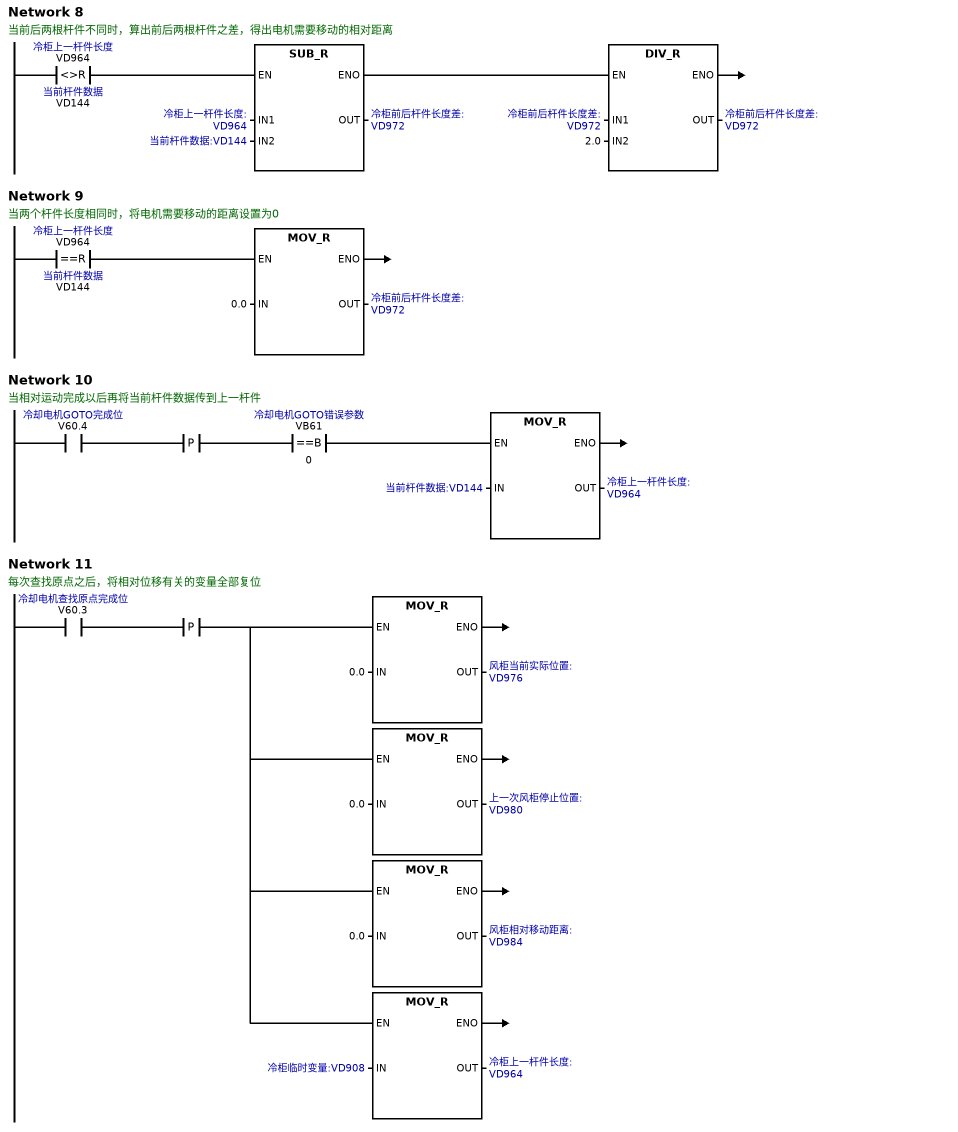
[picture p24: SBR16 networks 8-11]
Network 8
// 当前后两根杆件不同时，算出前后两根杆件之差，得出电机需要移动的相对距离
LDR<>  冷柜上一杆件长度:VD964, 当前杆件数据:VD144
MOVR   冷柜上一杆件长度:VD964, 冷柜前后杆件长度差:VD972
AENO
-R     当前杆件数据:VD144, 冷柜前后杆件长度差:VD972
AENO
/R     2.0, 冷柜前后杆件长度差:VD972
Network 9
// 当两个杆件长度相同时，将电机需要移动的距离设置为0
LDR=   冷柜上一杆件长度:VD964, 当前杆件数据:VD144
MOVR   0.0, 冷柜前后杆件长度差:VD972
Network 10
// 当相对运动完成以后再将当前杆件数据传到上一杆件
LD     冷却电机GOTO完成位:V60.4
EU
AB=    冷却电机GOTO错误参数:VB61, 0
MOVR   当前杆件数据:VD144, 冷柜上一杆件长度:VD964
Network 11
// 每次查找原点之后，将相对位移有关的变量全部复位
LD     冷却电机查找原点完成位:V60.3
EU
MOVR   0.0, 风柜当前实际位置:VD976
MOVR   0.0, 上一次风柜停止位置:VD980
MOVR   0.0, 风柜相对移动距离:VD984
MOVR   冷柜临时变量:VD908, 冷柜上一杆件长度:VD964
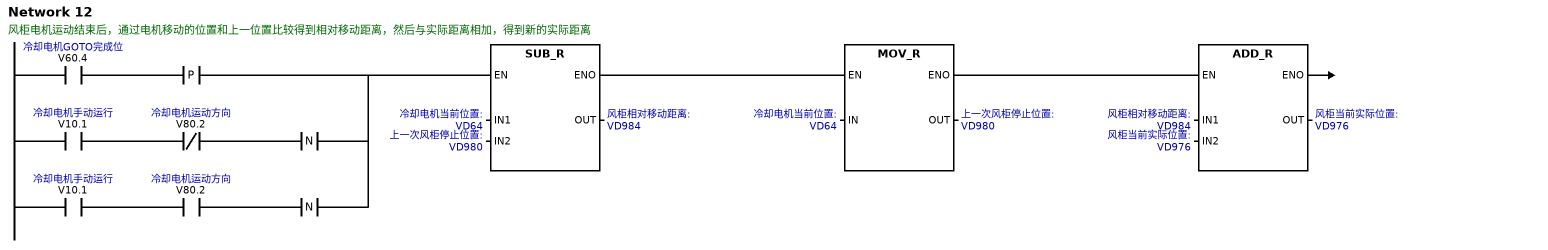
Network 12
// 风柜电机运动结束后，通过电机移动的位置和上一位置比较得到相对移动距离，然后与实际距离相加，得到新的实际距离
LD     冷却电机GOTO完成位:V60.4
EU
LD     冷却电机手动运行:V10.1
AN     冷却电机运动方向:V80.2
ED
OLD
LD     冷却电机手动运行:V10.1
A      冷却电机运动方向:V80.2
ED
OLD
MOVR   冷却电机当前位置:VD64, 风柜相对移动距离:VD984
AENO
-R     上一次风柜停止位置:VD980, 风柜相对移动距离:VD984
AENO
MOVR   冷却电机当前位置:VD64, 上一次风柜停止位置:VD980
AENO
+R     风柜相对移动距离:VD984, 风柜当前实际位置:VD976
END_SUBROUTINE_BLOCK

SUBROUTINE_BLOCK 冷却电机手动控制:SBR18
TITLE=子程序注释
BEGIN
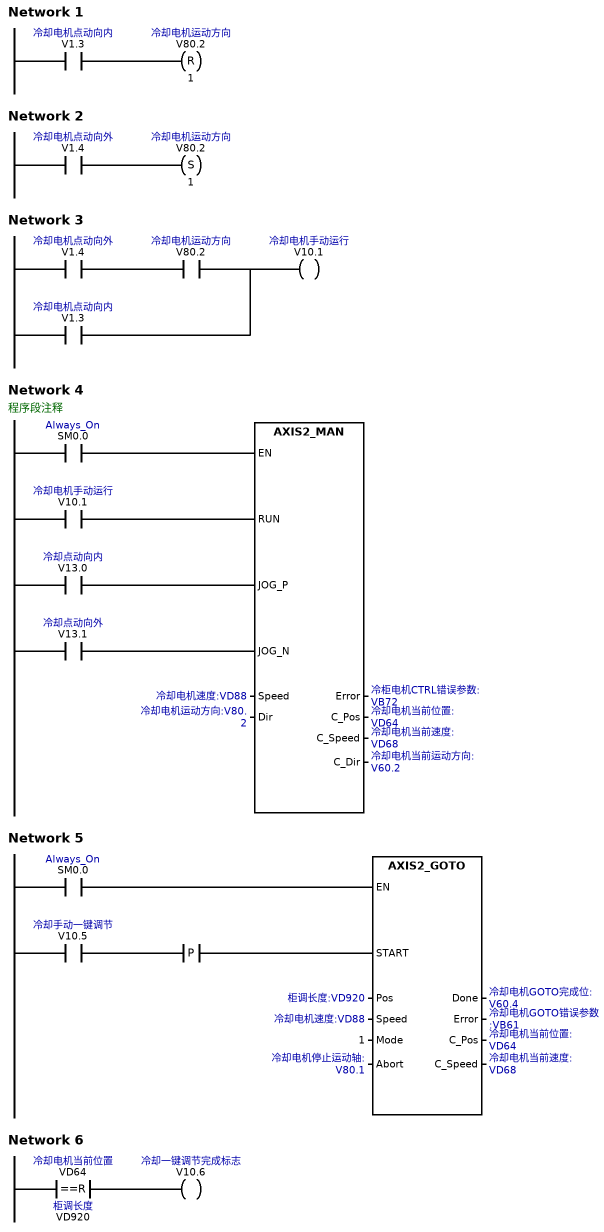
Network 1
LD     冷却电机点动向内:V1.3
R      冷却电机运动方向:V80.2, 1
Network 2
LD     冷却电机点动向外:V1.4
S      冷却电机运动方向:V80.2, 1
Network 3
LD     冷却电机点动向外:V1.4
A      冷却电机运动方向:V80.2
O      冷却电机点动向内:V1.3
=      冷却电机手动运行:V10.1
Network 4
// 程序段注释
LD     Always_On:SM0.0
=      L60.0
LD     冷却电机手动运行:V10.1
=      L63.7
LD     冷却点动向内:V13.0
=      L63.6
LD     冷却点动向外:V13.1
=      L63.5
LD     L60.0
CALL   AXIS2_MAN:SBR11, L63.7, L63.6, L63.5, 冷却电机速度:VD88, 冷却电机运动方向:V80.2, 冷柜电机CTRL错误参数:VB72, 冷却电机当前位置:VD64, 冷却电机当前速度:VD68, 冷却电机当前运动方向:V60.2
Network 5
LD     Always_On:SM0.0
=      L60.0
LD     冷却手动一键调节:V10.5
EU
=      L63.7
LD     L60.0
CALL   AXIS2_GOTO:SBR12, L63.7, 柜调长度:VD920, 冷却电机速度:VD88, 1, 冷却电机停止运动轴:V80.1, 冷却电机GOTO完成位:V60.4, 冷却电机GOTO错误参数:VB61, 冷却电机当前位置:VD64, 冷却电机当前速度:VD68
Network 6
LDR=   冷却电机当前位置:VD64, 柜调长度:VD920
=      冷却一键调节完成标志:V10.6
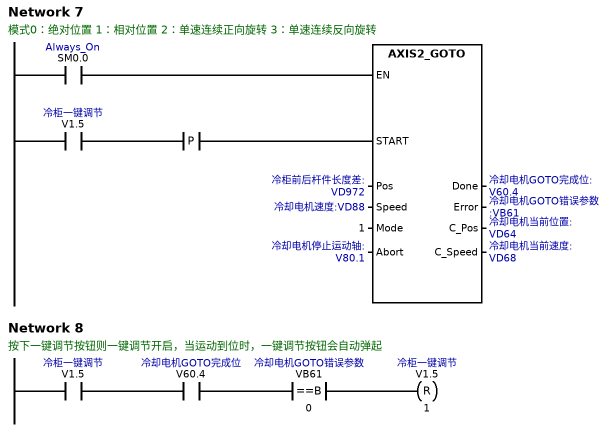
Network 7
// 模式0：绝对位置 1：相对位置 2：单速连续正向旋转 3：单速连续反向旋转
LD     Always_On:SM0.0
=      L60.0
LD     冷柜一键调节:V1.5
EU
=      L63.7
LD     L60.0
CALL   AXIS2_GOTO:SBR12, L63.7, 冷柜前后杆件长度差:VD972, 冷却电机速度:VD88, 1, 冷却电机停止运动轴:V80.1, 冷却电机GOTO完成位:V60.4, 冷却电机GOTO错误参数:VB61, 冷却电机当前位置:VD64, 冷却电机当前速度:VD68
Network 8
// 按下一键调节按钮则一键调节开启，当运动到位时，一键调节按钮会自动弹起
LD     冷柜一键调节:V1.5
A      冷却电机GOTO完成位:V60.4
AB=    冷却电机GOTO错误参数:VB61, 0
R      冷柜一键调节:V1.5, 1
END_SUBROUTINE_BLOCK

SUBROUTINE_BLOCK 链传动电机控制:SBR19
TITLE=子程序注释
BEGIN
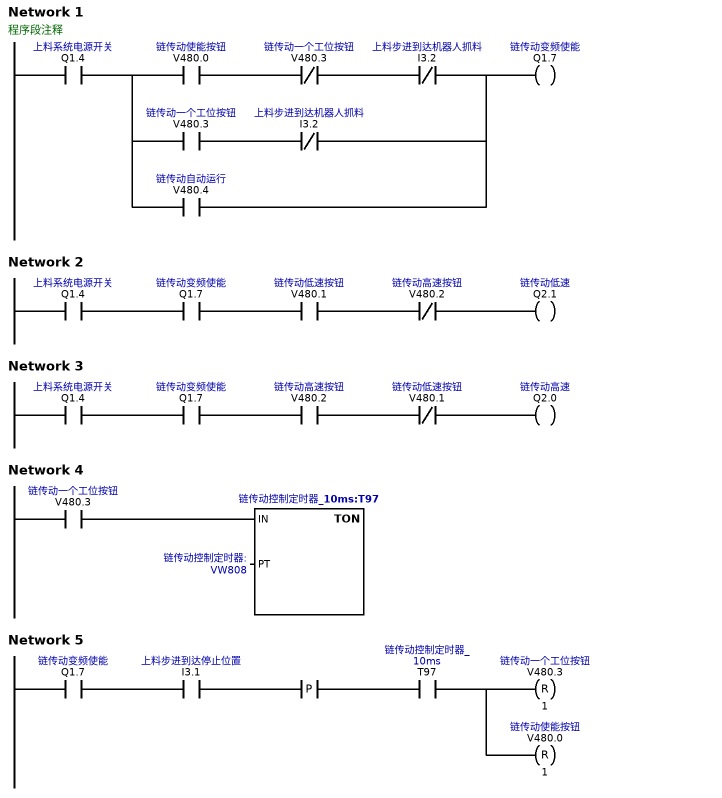
Network 1
// 程序段注释
LD     上料系统电源开关:Q1.4
LD     链传动使能按钮:V480.0
AN     链传动一个工位按钮:V480.3
AN     上料步进到达机器人抓料:I3.2
LD     链传动一个工位按钮:V480.3
AN     上料步进到达机器人抓料:I3.2
OLD
O      链传动自动运行:V480.4
ALD
=      链传动变频使能:Q1.7
Network 2
LD     上料系统电源开关:Q1.4
A      链传动变频使能:Q1.7
A      链传动低速按钮:V480.1
AN     链传动高速按钮:V480.2
=      链传动低速:Q2.1
Network 3
LD     上料系统电源开关:Q1.4
A      链传动变频使能:Q1.7
A      链传动高速按钮:V480.2
AN     链传动低速按钮:V480.1
=      链传动高速:Q2.0
Network 4
LD     链传动一个工位按钮:V480.3
TON    链传动控制定时器_10ms:T97, 链传动控制定时器:VW808
Network 5
LD     链传动变频使能:Q1.7
A      上料步进到达停止位置:I3.1
EU
A      链传动控制定时器_10ms:T97
R      链传动一个工位按钮:V480.3, 1
R      链传动使能按钮:V480.0, 1
END_SUBROUTINE_BLOCK

SUBROUTINE_BLOCK 数据初始化:SBR20
TITLE=子程序注释
BEGIN
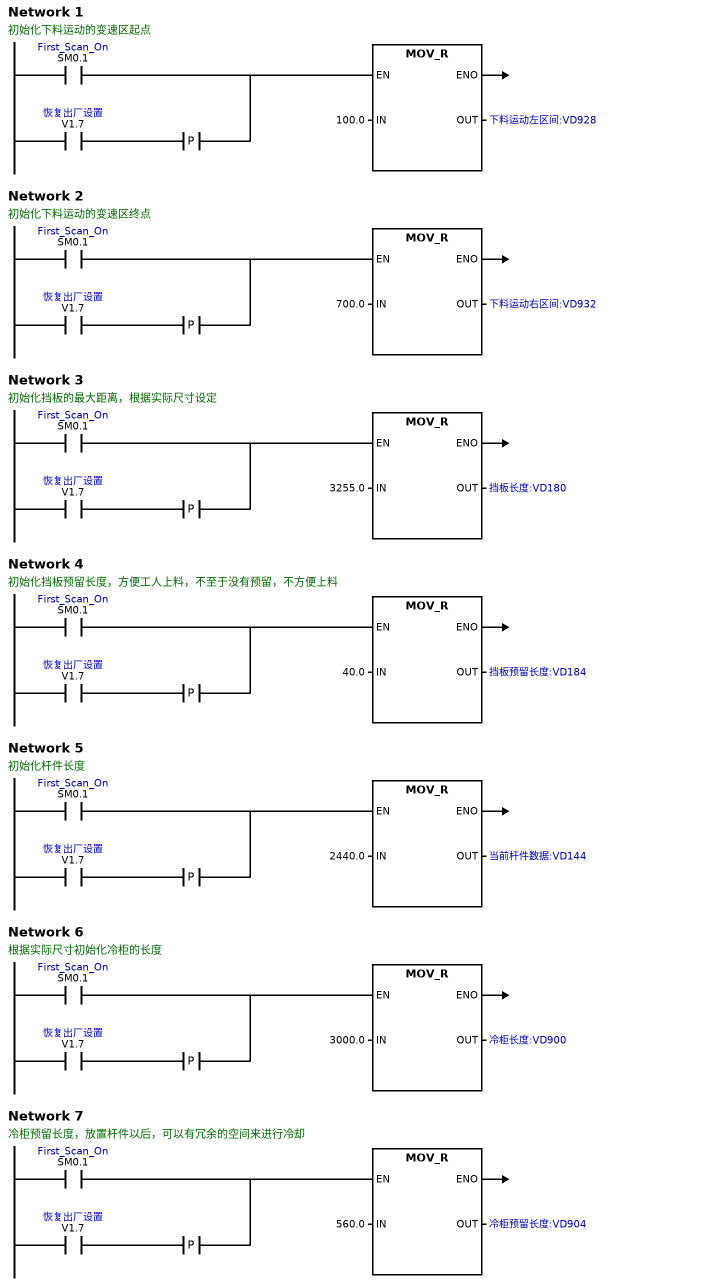
Network 1
// 初始化下料运动的变速区起点
LD     First_Scan_On:SM0.1
LD     恢复出厂设置:V1.7
EU
OLD
MOVR   100.0, 下料运动左区间:VD928
Network 2
// 初始化下料运动的变速区终点
LD     First_Scan_On:SM0.1
LD     恢复出厂设置:V1.7
EU
OLD
MOVR   700.0, 下料运动右区间:VD932
Network 3
// 初始化挡板的最大距离，根据实际尺寸设定
LD     First_Scan_On:SM0.1
LD     恢复出厂设置:V1.7
EU
OLD
MOVR   3255.0, 挡板长度:VD180
Network 4
// 初始化挡板预留长度，方便工人上料，不至于没有预留，不方便上料
LD     First_Scan_On:SM0.1
LD     恢复出厂设置:V1.7
EU
OLD
MOVR   40.0, 挡板预留长度:VD184
Network 5
// 初始化杆件长度
LD     First_Scan_On:SM0.1
LD     恢复出厂设置:V1.7
EU
OLD
MOVR   2440.0, 当前杆件数据:VD144
Network 6
// 根据实际尺寸初始化冷柜的长度
LD     First_Scan_On:SM0.1
LD     恢复出厂设置:V1.7
EU
OLD
MOVR   3000.0, 冷柜长度:VD900
Network 7
// 冷柜预留长度，放置杆件以后，可以有冗余的空间来进行冷却
LD     First_Scan_On:SM0.1
LD     恢复出厂设置:V1.7
EU
OLD
MOVR   560.0, 冷柜预留长度:VD904
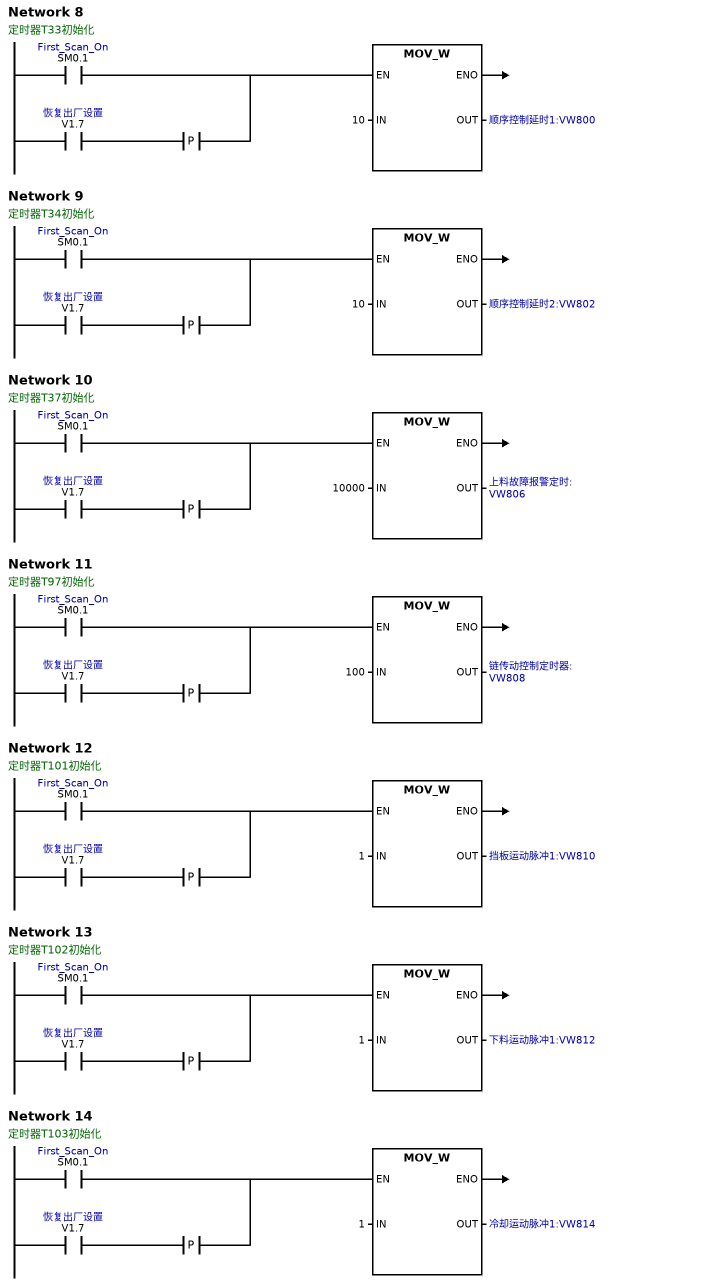
Network 8
// 定时器T33初始化
LD     First_Scan_On:SM0.1
LD     恢复出厂设置:V1.7
EU
OLD
MOVW   10, 顺序控制延时1:VW800
Network 9
// 定时器T34初始化
LD     First_Scan_On:SM0.1
LD     恢复出厂设置:V1.7
EU
OLD
MOVW   10, 顺序控制延时2:VW802
Network 10
// 定时器T37初始化
LD     First_Scan_On:SM0.1
LD     恢复出厂设置:V1.7
EU
OLD
MOVW   10000, 上料故障报警定时:VW806
Network 11
// 定时器T97初始化
LD     First_Scan_On:SM0.1
LD     恢复出厂设置:V1.7
EU
OLD
MOVW   100, 链传动控制定时器:VW808
Network 12
// 定时器T101初始化
LD     First_Scan_On:SM0.1
LD     恢复出厂设置:V1.7
EU
OLD
MOVW   1, 挡板运动脉冲1:VW810
Network 13
// 定时器T102初始化
LD     First_Scan_On:SM0.1
LD     恢复出厂设置:V1.7
EU
OLD
MOVW   1, 下料运动脉冲1:VW812
Network 14
// 定时器T103初始化
LD     First_Scan_On:SM0.1
LD     恢复出厂设置:V1.7
EU
OLD
MOVW   1, 冷却运动脉冲1:VW814
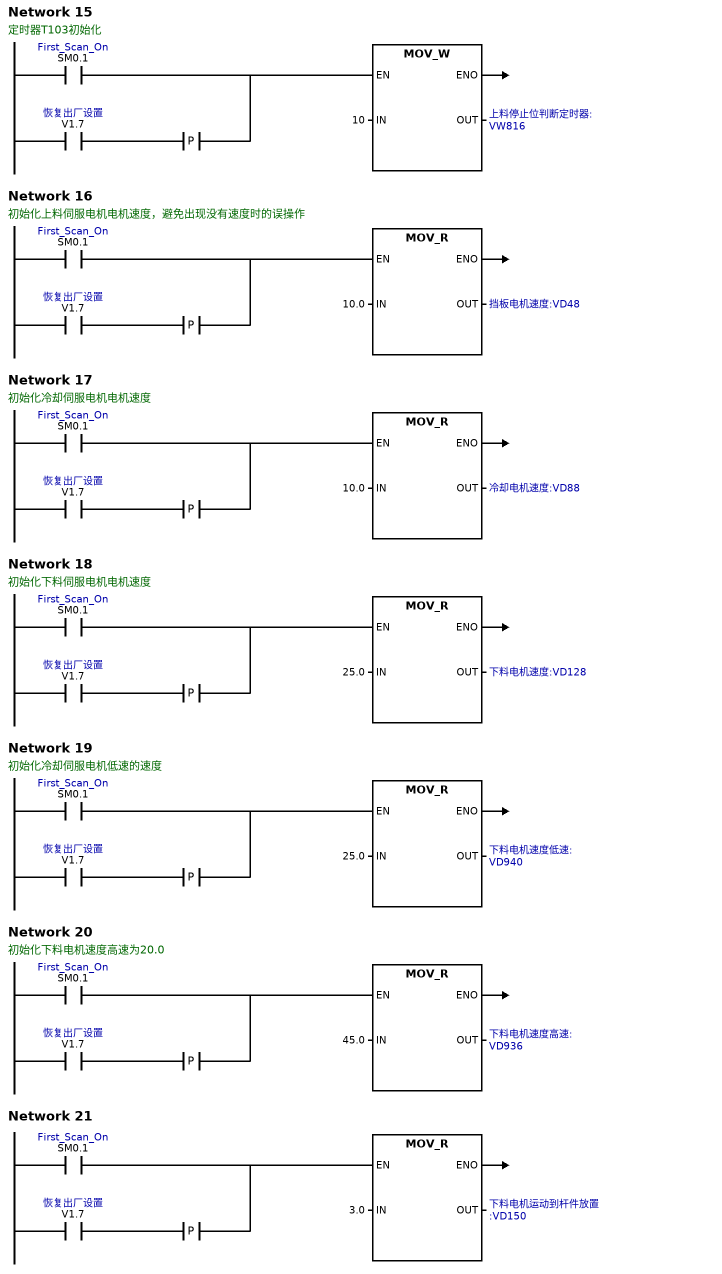
Network 15
// 定时器T103初始化
LD     First_Scan_On:SM0.1
LD     恢复出厂设置:V1.7
EU
OLD
MOVW   10, 上料停止位判断定时器:VW816
Network 16
// 初始化上料伺服电机电机速度，避免出现没有速度时的误操作
LD     First_Scan_On:SM0.1
LD     恢复出厂设置:V1.7
EU
OLD
MOVR   10.0, 挡板电机速度:VD48
Network 17
// 初始化冷却伺服电机电机速度
LD     First_Scan_On:SM0.1
LD     恢复出厂设置:V1.7
EU
OLD
MOVR   10.0, 冷却电机速度:VD88
Network 18
// 初始化下料伺服电机电机速度
LD     First_Scan_On:SM0.1
LD     恢复出厂设置:V1.7
EU
OLD
MOVR   25.0, 下料电机速度:VD128
Network 19
// 初始化冷却伺服电机低速的速度
LD     First_Scan_On:SM0.1
LD     恢复出厂设置:V1.7
EU
OLD
MOVR   25.0, 下料电机速度低速:VD940
Network 20
// 初始化下料电机速度高速为20.0
LD     First_Scan_On:SM0.1
LD     恢复出厂设置:V1.7
EU
OLD
MOVR   45.0, 下料电机速度高速:VD936
Network 21
LD     First_Scan_On:SM0.1
LD     恢复出厂设置:V1.7
EU
OLD
MOVR   3.0, 下料电机运动到杆件放置:VD150
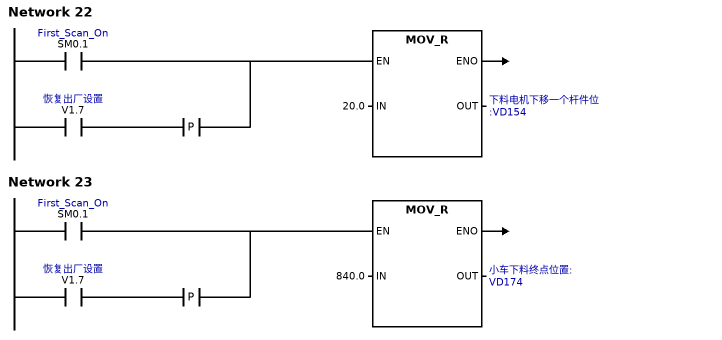
Network 22
LD     First_Scan_On:SM0.1
LD     恢复出厂设置:V1.7
EU
OLD
MOVR   20.0, 下料电机下移一个杆件位:VD154
Network 23
LD     First_Scan_On:SM0.1
LD     恢复出厂设置:V1.7
EU
OLD
MOVR   840.0, 小车下料终点位置:VD174
END_SUBROUTINE_BLOCK

SUBROUTINE_BLOCK 故障报警:SBR21
TITLE=子程序注释
BEGIN
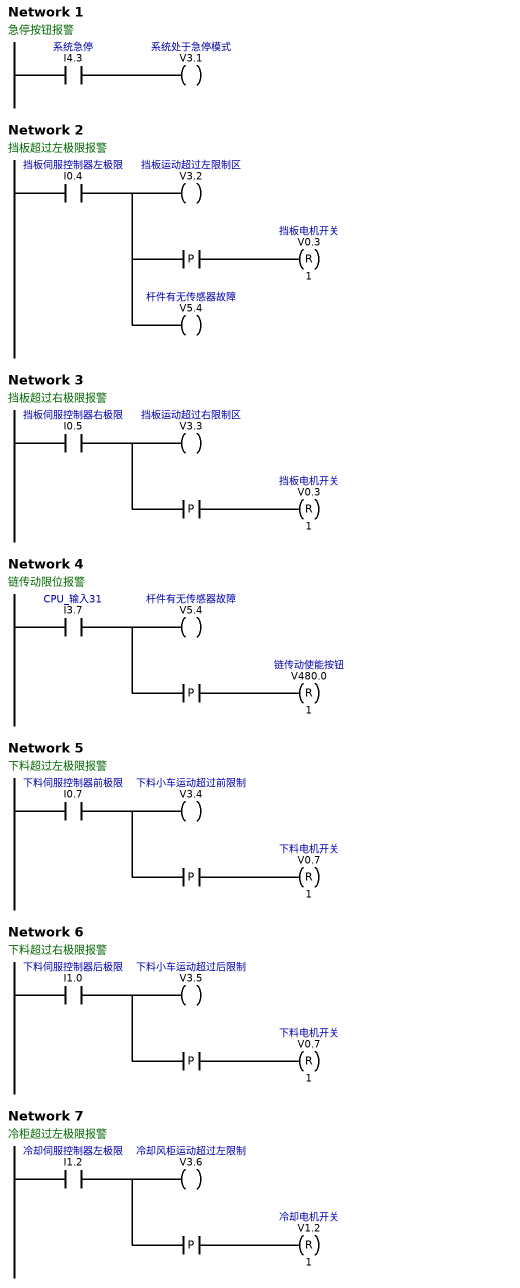
Network 1
// 急停按钮报警
LD     系统急停:I4.3
=      系统处于急停模式:V3.1
Network 2
// 挡板超过左极限报警
LD     挡板伺服控制器左极限:I0.4
LPS
=      挡板运动超过左限制区:V3.2
EU
R      挡板电机开关:V0.3, 1
LPP
=      杆件有无传感器故障:V5.4
Network 3
// 挡板超过右极限报警
LD     挡板伺服控制器右极限:I0.5
=      挡板运动超过右限制区:V3.3
EU
R      挡板电机开关:V0.3, 1
Network 4
// 链传动限位报警
LD     CPU_输入31:I3.7
=      杆件有无传感器故障:V5.4
EU
R      链传动使能按钮:V480.0, 1
Network 5
// 下料超过左极限报警
LD     下料伺服控制器前极限:I0.7
=      下料小车运动超过前限制:V3.4
EU
R      下料电机开关:V0.7, 1
Network 6
// 下料超过右极限报警
LD     下料伺服控制器后极限:I1.0
=      下料小车运动超过后限制:V3.5
EU
R      下料电机开关:V0.7, 1
Network 7
// 冷柜超过左极限报警
LD     冷却伺服控制器左极限:I1.2
=      冷却风柜运动超过左限制:V3.6
EU
R      冷却电机开关:V1.2, 1
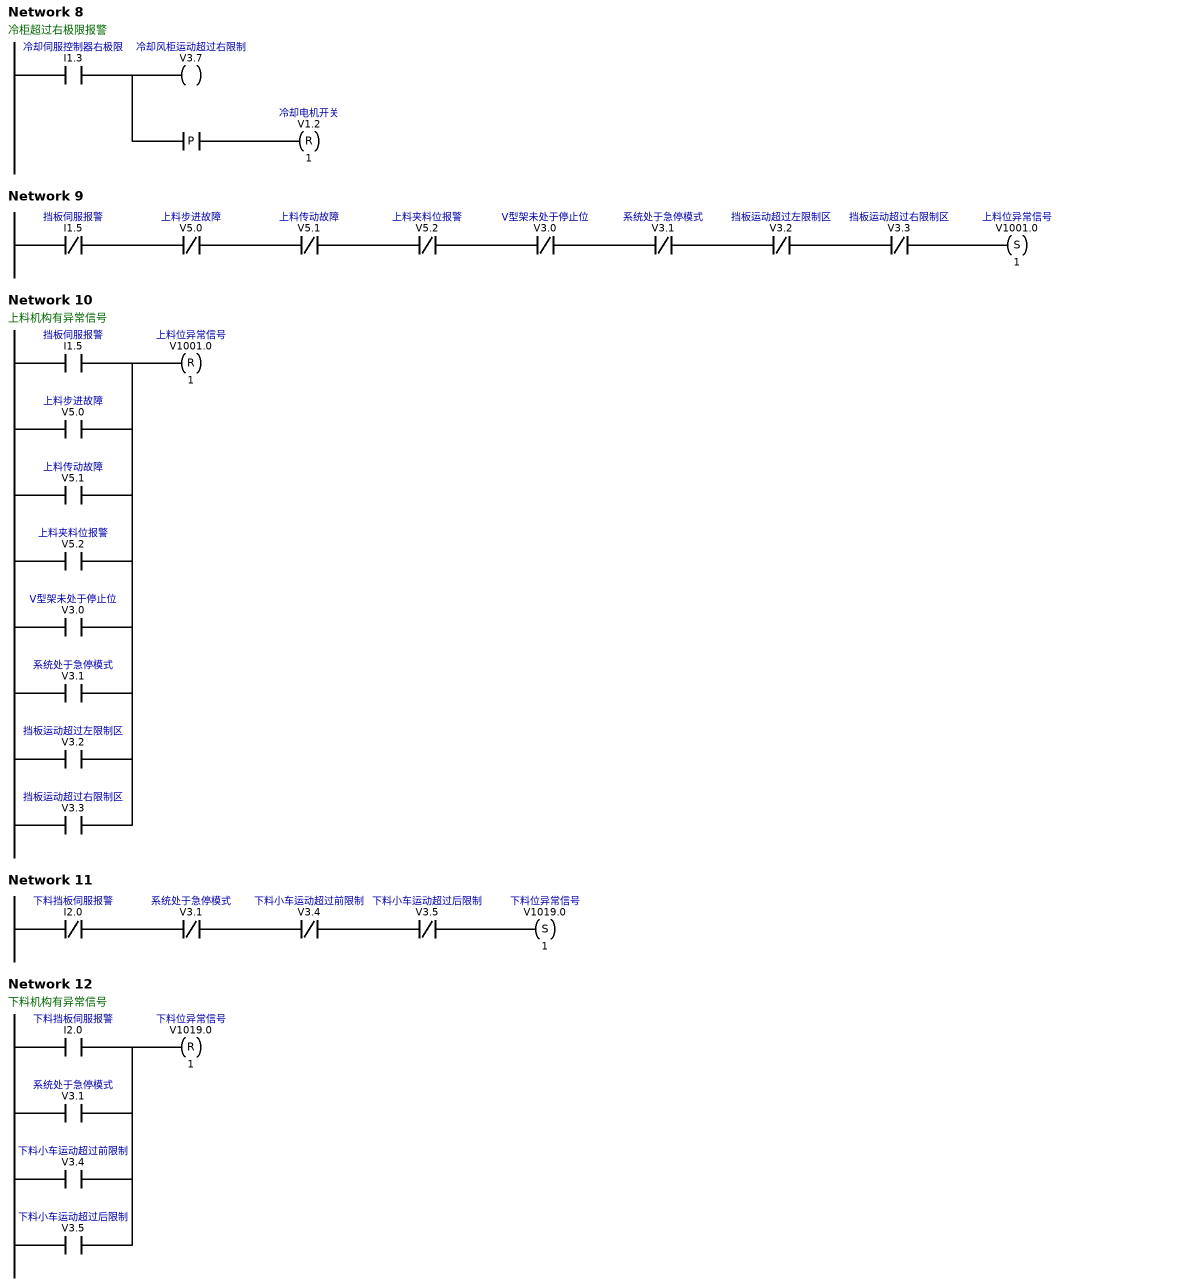
Network 8
// 冷柜超过右极限报警
LD     冷却伺服控制器右极限:I1.3
=      冷却风柜运动超过右限制:V3.7
EU
R      冷却电机开关:V1.2, 1
Network 9
LDN    挡板伺服报警:I1.5
AN     上料步进故障:V5.0
AN     上料传动故障:V5.1
AN     上料夹料位报警:V5.2
AN     V型架未处于停止位:V3.0
AN     系统处于急停模式:V3.1
AN     挡板运动超过左限制区:V3.2
AN     挡板运动超过右限制区:V3.3
S      上料位异常信号:V1001.0, 1
Network 10
// 上料机构有异常信号
LD     挡板伺服报警:I1.5
O      上料步进故障:V5.0
O      上料传动故障:V5.1
O      上料夹料位报警:V5.2
O      V型架未处于停止位:V3.0
O      系统处于急停模式:V3.1
O      挡板运动超过左限制区:V3.2
O      挡板运动超过右限制区:V3.3
R      上料位异常信号:V1001.0, 1
Network 11
LDN    下料挡板伺服报警:I2.0
AN     系统处于急停模式:V3.1
AN     下料小车运动超过前限制:V3.4
AN     下料小车运动超过后限制:V3.5
S      下料位异常信号:V1019.0, 1
Network 12
// 下料机构有异常信号
LD     下料挡板伺服报警:I2.0
O      系统处于急停模式:V3.1
O      下料小车运动超过前限制:V3.4
O      下料小车运动超过后限制:V3.5
R      下料位异常信号:V1019.0, 1
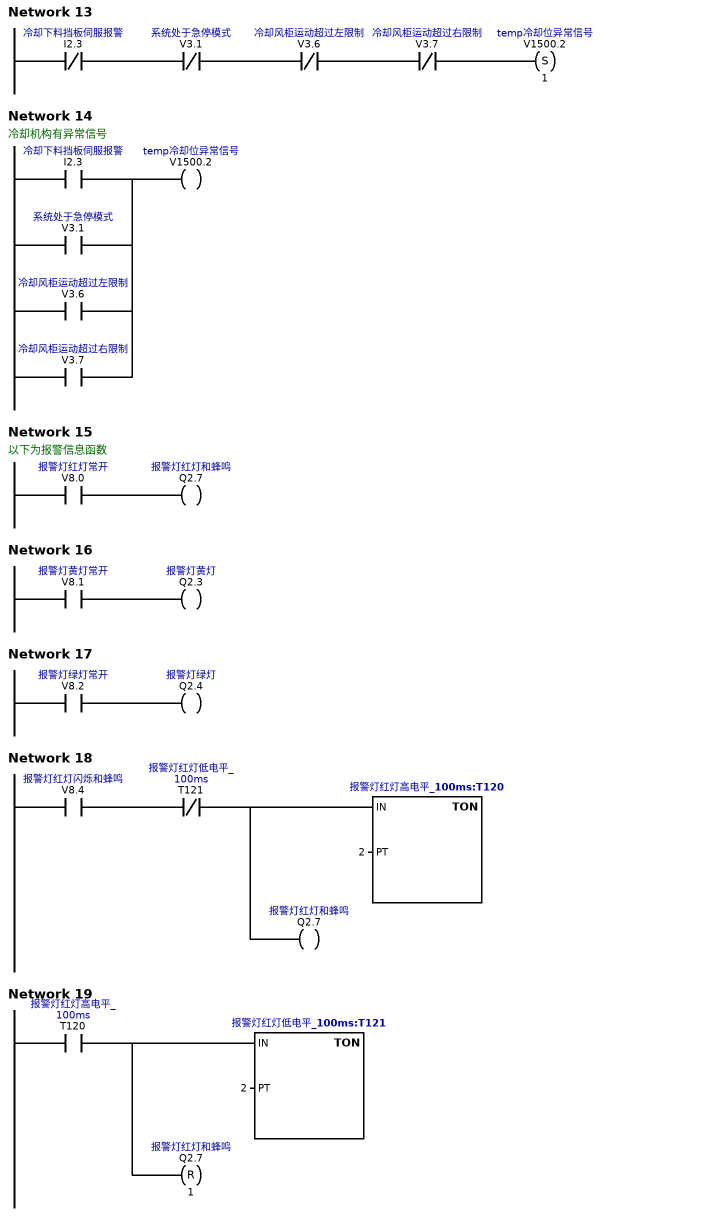
Network 13
LDN    冷却下料挡板伺服报警:I2.3
AN     系统处于急停模式:V3.1
AN     冷却风柜运动超过左限制:V3.6
AN     冷却风柜运动超过右限制:V3.7
S      temp冷却位异常信号:V1500.2, 1
Network 14
// 冷却机构有异常信号
LD     冷却下料挡板伺服报警:I2.3
O      系统处于急停模式:V3.1
O      冷却风柜运动超过左限制:V3.6
O      冷却风柜运动超过右限制:V3.7
=      temp冷却位异常信号:V1500.2
Network 15
// 以下为报警信息函数
LD     报警灯红灯常开:V8.0
=      报警灯红灯和蜂鸣:Q2.7
Network 16
LD     报警灯黄灯常开:V8.1
=      报警灯黄灯:Q2.3
Network 17
LD     报警灯绿灯常开:V8.2
=      报警灯绿灯:Q2.4
Network 18
LD     报警灯红灯闪烁和蜂鸣:V8.4
AN     报警灯红灯低电平_100ms:T121
TON    报警灯红灯高电平_100ms:T120, 2
=      报警灯红灯和蜂鸣:Q2.7
Network 19
LD     报警灯红灯高电平_100ms:T120
TON    报警灯红灯低电平_100ms:T121, 2
R      报警灯红灯和蜂鸣:Q2.7, 1
END_SUBROUTINE_BLOCK
